FUNCTION_BLOCK Port (* Service Interface Function Block Type *)
  (* Standard: 61499-2; Description: Copyright (c) 2021, 2022 Jonathan Lainer This program and the accompanying materials are made available under the terms of the Eclipse Public License 2.0 which is available at https://www.eclipse.org/legal/epl-2.0/ SPDX-License-Identifier: EPL-2.0 *)
  (* Version 1.0, 2021-02-22, Jonathan Lainer, Initial Contribution *)
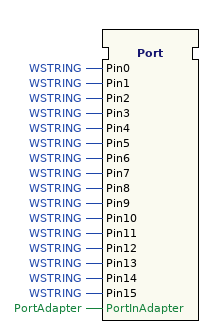
  VAR_INPUT
    Pin0 : WSTRING; (* Name of the Pin *)
    Pin1 : WSTRING; (* Name of the Pin *)
    Pin2 : WSTRING; (* Name of the Pin *)
    Pin3 : WSTRING; (* Name of the Pin *)
    Pin4 : WSTRING; (* Name of the Pin *)
    Pin5 : WSTRING; (* Name of the Pin *)
    Pin6 : WSTRING; (* Name of the Pin *)
    Pin7 : WSTRING; (* Name of the Pin *)
    Pin8 : WSTRING; (* Name of the Pin *)
    Pin9 : WSTRING; (* Name of the Pin *)
    Pin10 : WSTRING; (* Name of the Pin *)
    Pin11 : WSTRING; (* Name of the Pin *)
    Pin12 : WSTRING; (* Name of the Pin *)
    Pin13 : WSTRING; (* Name of the Pin *)
    Pin14 : WSTRING; (* Name of the Pin *)
    Pin15 : WSTRING; (* Name of the Pin *)
  END_VAR
  SOCKETS
    PortInAdapter : PortAdapter;
  END_SOCKETS
  SERVICE APPLICATION/RESOURCE (* Service Interface Function Block Type *)
    SEQUENCE normal_establishment
      APPLICATION.INIT+(PARAMS) -> RESOURCE.initialize(PARAMS) -> APPLICATION.INITO+();
    END_SEQUENCE
    SEQUENCE unsuccessful_establishment
      APPLICATION.INIT+(PARAMS) -> RESOURCE.initialize(PARAMS) -> APPLICATION.INITO-(STATUS);
    END_SEQUENCE
    SEQUENCE request_confirm
      APPLICATION.REQ+(SD) -> RESOURCE.request(SD) -> APPLICATION.CNF+(RD);
    END_SEQUENCE
    SEQUENCE request_inhibited
      APPLICATION.REQ-(SD) -> APPLICATION.CNF-(STATUS);
    END_SEQUENCE
    SEQUENCE request_error
      APPLICATION.REQ+(SD) -> RESOURCE.request(SD) -> APPLICATION.CNF-(STATUS);
    END_SEQUENCE
    SEQUENCE indication_response
      RESOURCE.indicate(RD) -> APPLICATION.IND+(RD);
      APPLICATION.RSP(QI,SD) -> RESOURCE.response(QI,SD);
    END_SEQUENCE
    SEQUENCE indication_inhibited
      RESOURCE.indicate(RD,QI=FALSE) -> RESOURCE.inhibited();
    END_SEQUENCE
    SEQUENCE error_indication
      RESOURCE.error(STATUS) -> APPLICATION.IND-(STATUS);
    END_SEQUENCE
    SEQUENCE application_initiated_termination
      APPLICATION.INIT-() -> RESOURCE.terminate() -> APPLICATION.INITO-(STATUS);
    END_SEQUENCE
    SEQUENCE resource_initiated_termination
      -> APPLICATION.INITO-(STATUS);
    END_SEQUENCE
  END_SERVICE
END_FUNCTION_BLOCK
